Universal Robots PolyScope program: Hospital_big_top.urp

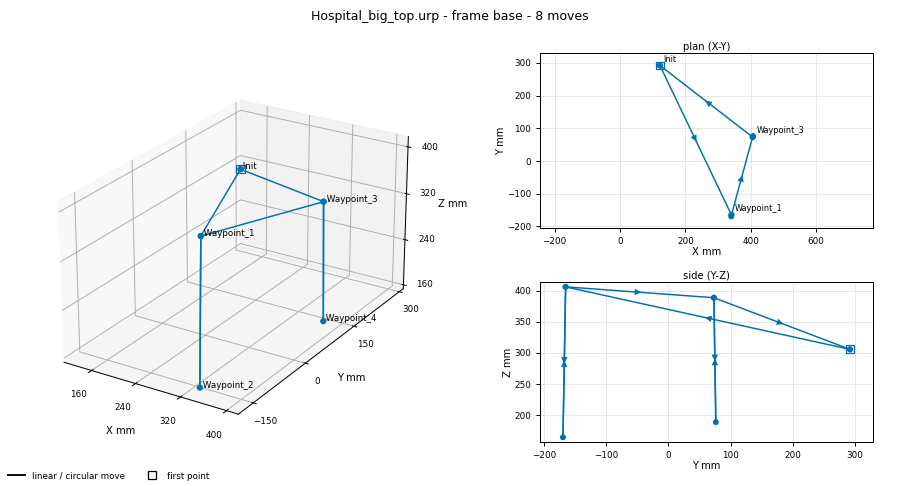
[picture p0: tool path of Hospital_big_top.urp in frame base, 8 of 8 moves have a stored position in this frame; points joined in program order, loops and branches not executed]
Program Hospital_big_top (installation=default directory=/programs/Mursal createdIn=5.11.11.1010533 lastSavedIn=5.11.11.1010533 robotSerialNumber=20205300864)
Calibrated DH parameters: a=[-0.000166, -0.243494, -0.153108, 0.000057, -0.000123, 0]; d=[0.151897, -1.34267, 53.988124, -52.514559, 0.085283, 0.092193]; alpha=[1.572472, -0.003756, 0.002824, 1.570807, -1.572621, 0]; deltaTheta=[0, 0.020704, 7.033215, -0.770746, 0.000004, 0]
Robot Program (runOnlyOnce=true)
  MoveL speed 250 mm/s, acceleration 1200 mm/s^2 (useActiveTCP=true) feature=Base
    Waypoint Init: TCP in base x=122.111 y=292.108 z=305.716 mm, rx=1.1347 ry=-2.9295 rz=0.0001 rad; joints [91.642, -87.585, -91.769, -90.545, 90.032, 859.396] deg
    Waypoint Waypoint_1: TCP in base x=340.922 y=-165.039 z=406.176 mm, rx=-2.2707 ry=2.171 rz=-0.0001 rad; joints [-5.588, -113.056, -31.918, -124.915, 89.852, 711.883] deg
    Waypoint Waypoint_2: TCP in base x=340.1 y=-169.331 z=164.432 mm, rx=-2.2706 ry=2.171 rz=-0.0001 rad; joints [-6.442, -112.908, -101.237, -55.744, 89.984, 711.162] deg
    URCap Gripper (Robotiq_Grippers, Robotiq Inc.) dataModel(position=100.0, force=9.0, speed=0.0, positionInDouble=100.0, forceInDouble=9.0, speedInDouble=0.0, slaveIds=[9], blocking=true, robotCompliant=false)
    Waypoint Waypoint_1: TCP in base x=340.922 y=-165.039 z=406.176 mm, rx=-2.2707 ry=2.171 rz=-0.0001 rad; joints [-5.588, -113.056, -31.918, -124.915, 89.852, 711.883] deg
    Waypoint Waypoint_3: TCP in base x=405.589 y=73.278 z=388.751 mm, rx=3.1407 ry=0.0712 rz=0 rad; joints [28.801, -122.956, -21.226, -125.714, 89.817, 656.227] deg
    Waypoint Waypoint_4: TCP in base x=406.944 y=76.371 z=188.837 mm, rx=3.1415 ry=0.013 rz=0.0001 rad; joints [28.955, -117.561, -86.466, -65.868, 89.957, 658.617] deg
    URCap Gripper (Robotiq_Grippers, Robotiq Inc.) dataModel(position=0.0, force=9.0, speed=0.0, positionInDouble=0.0, forceInDouble=9.0, speedInDouble=0.0, slaveIds=[9], blocking=true, robotCompliant=false)
    Waypoint Waypoint_3: TCP in base x=405.589 y=73.278 z=388.751 mm, rx=3.1407 ry=0.0712 rz=0 rad; joints [28.801, -122.956, -21.226, -125.714, 89.817, 656.227] deg
    Waypoint Init: TCP in base x=122.111 y=292.108 z=305.716 mm, rx=1.1347 ry=-2.9295 rz=0.0001 rad; joints [91.642, -87.585, -91.769, -90.545, 90.032, 859.396] deg
